INTERFACE ITF_Regelschuif_In_DG

METHOD get : SINT
VAR_INPUT
END_VAR
END_METHOD

END_INTERFACE

(* stored: Version 1.1.0.1, ProductVersion 3.1.4026.8
   Itf ITF_Regelschuif_In_DG: Id {47c62877-1ab7-47f7-b1c3-92bbb8e1350c}
   Method get: Id {294a86c7-d225-425c-a33c-058e3dcf1668} *)
